{attribute 'linkalways'} 
{attribute 'no_explicit_call' := 'This FB is a CLASS and must be accessed using methods or properties'}
{attribute 'enable_dynamic_creation'}
FUNCTION_BLOCK Node_F_VN_MedianElementElementwise_TcVnVector2_INT EXTENDS VisionNode
VAR
    ipContainer : _ITcVnContainer;
    aMedian : _TcVnVector2_INT;
    hrPrev : _HRESULT(S_OK);
    hresult : _HRESULT(S_OK);
END_VAR

METHOD PUBLIC  Clone : I_Node
VAR
	pNode : POINTER TO Node_F_VN_MedianElementElementwise_TcVnVector2_INT;
END_VAR
pNode := __NEW(Node_F_VN_MedianElementElementwise_TcVnVector2_INT);
Clone := pNode^;
END_METHOD

METHOD FB_init : BOOL
VAR_INPUT
	bInitRetains : BOOL; // if TRUE, the retain variables are initialized (warm start / cold start)
	bInCopyCode : BOOL;  // if TRUE, the instance afterwards gets moved into the copy code (online change)
END_VAR
AddInput('ipContainer', ipContainer);
AddInput('hrPrev', hrPrev);
AddOutput('ipContainer', ipContainer);
AddOutput('aMedian', aMedian);
AddOutput('hresult',hresult);
END_METHOD

METHOD PROTECTED OnExecute
hresult.Value := F_VN_MedianElementElementwise_TcVnVector2_INT(
    ipContainer := ipContainer.Value,
    aMedian := aMedian.Value,
    hrPrev:= hrPrev.Value);
END_METHOD

METHOD PUBLIC PreExecutionCheck
VAR_INPUT
	Check : I_PreExecutionChecks;
END_VAR
Check.IsTrue(ipContainer.IsValid, 'ipContainer must be a valid container');
Check.IsTrue(ipContainer.IsType(TC_GLOBAL_CONST_LIST.ContainerType_Vector_TcVnVector2_INT), 'ipContainer contains incorrect type');
END_METHOD

END_FUNCTION_BLOCK

(* stored: Version 1.1.0.1, ProductVersion 3.1.4026.13
   POU Node_F_VN_MedianElementElementwise_TcVnVector2_INT: Id {aa162ef7-7b75-4132-87df-28ce6c70b932}, SpecialFunc None
   Folder Constructor: Id {28e4cdbd-b909-4f87-8d98-55d6a6facced}
   Method Clone: Id {1283b373-dae6-4bf8-ac9c-11c9061610c9}
   Method FB_init: Id {4da293fd-1a33-42f1-bf9c-39871abfc19e}
   Method OnExecute: Id {3c763f0e-01c5-4fde-a651-e6caf7d74d40}
   Method PreExecutionCheck: Id {d636acae-e67b-4086-994e-b3309d0ae5ba} *)
